PROGRAM Pneumatic_Axis
VAR
    fbPneumaticAxis : FB_PneumaticAxis;

    stPneumaticAxisStruct: INT;
    stPneumaticAxisInputs: INT;
END_VAR

fbPneumaticAxis();

END_PROGRAM

(* stored: Version 1.1.0.1, ProductVersion 3.1.4024.5
   POU Pneumatic_Axis: Id {6b0fdf6b-27a8-416b-b2fa-fda7ea3fc6bb}, SpecialFunc None *)
